{attribute 'conditionalshow'}
FUNCTION_BLOCK FB_GantryXYZ EXTENDS FB_PackML_BaseModule IMPLEMENTS I_GantryConfigProvider
VAR
	
	fbHomeMcQ           : MC_Home;
    // =========================================================
    //  DEPENDENCIES & SUB-MODULES
    // =========================================================
    _RecipeBuilder      : I_RecipeBuilder;
    ipSubModules_Init   : ARRAY[1..Parameters_PackML_Base.MAX_NO_OF_SUBMODULES] OF I_PackML_BaseModule := [];

	ExecutorCutX 		: FB_Exec_Pneumatic_PTP;
	ExecutorCutY 		: FB_Exec_Pneumatic_PTP;	
	ExecutorGrooveXY	: FB_Exec_Spindle_PTP;
	ExecutorDrill 		: FB_Exec_Drill_PTP;
	ExecTangentialFeed	: FB_Exec_Tangential_FeedTable;
	
	ExecutorNCI 		: FB_Exec_Spindle_GCodeXYZ;
	
	_Limits : ST_GantryXYZ_Limits;


    // =========================================================
    //  HMI & COMMANDS
    // =========================================================
    GantryXYZ_HMI       : ST_GantryXYZ_HMI;
    _ProgramIdRequested : E_RecipeID;

    // =========================================================
    //  COMPONENTS (AXES & CYLINDERS)
    // =========================================================
    AxisX               : FB_Component_BasicAxis := (Name := 'AxisX');
    AxisY               : FB_Component_BasicAxis := (Name := 'AxisY');
    AxisZ               : FB_Component_BasicAxis := (Name := 'AxisZ');
	AxisQ               : FB_Component_BasicAxis := (Name := 'AxisQ Tangential'); 
	
	
	NciChannel          	: FB_NciChannel := (Name := 'NCI Channel 1');
	NciChannelTangential	: FB_NciChannelTangential := (Name := 'NCI Channel Tangential');
	
	
	
	// [Typ osi: 1=X, 2=Y, 3=Z] , [Typ profilu z Enuma]
	ProfilesX : ARRAY[E_MachineProfile.eHoming..E_MachineProfile.eManual] OF ST_AxisProfile;
	ProfilesY : ARRAY[E_MachineProfile.eHoming..E_MachineProfile.eManual] OF ST_AxisProfile;
	ProfilesZ : ARRAY[E_MachineProfile.eHoming..E_MachineProfile.eManual] OF ST_AxisProfile;
	ProfilesQ : ARRAY[E_MachineProfile.eHoming..E_MachineProfile.eManual] OF ST_AxisProfile;
	
	// Flagi określające typ napędu dla konkretnej osi (TRUE = SoE/AX5000, FALSE = CoE)
    AxisX_IsSoE : BOOL := FALSE;
    AxisY_IsSoE : BOOL := FALSE;
    AxisZ_IsSoE : BOOL := FALSE;
 
	CylinderCuttingX : FB_Cylinder := (Name := 'Cylinder X');
    CylinderCuttingY : FB_Cylinder := (Name := 'Cylinder Y');

    // =========================================================
    //  HOMING STRATEGIES
    // =========================================================
    fbHomeStratX        : FB_Homing_StandardNC;
    fbHomeStratY        : FB_Homing_StandardNC;
    fbHomeStratZ        : FB_Homing_StandardNC;
	fbHomeStratQ 		: FB_Homing_Direct;

    // =========================================================
    //  ALARMS
    // =========================================================
    GantryAlarms        : ARRAY[1..GANTRY_ALARM_COUNT] OF FB_TcAlarm;
	
	ResetStratX : FB_ResetRoutine_SoEDrive;
	ResetStratY : FB_ResetRoutine_SoEDrive;
	ResetStratZ : FB_ResetRoutine_SoEDrive;

END_VAR

VAR CONSTANT
    GANTRY_ALARM_COUNT  : INT := 5;
END_VAR

METHOD PROTECTED Aborting
VAR
    i               : UDINT;
    SubModulesReady : BOOL := TRUE;
END_VAR
VAR_INST
    AbortStepTimer  : TON; 
END_VAR
CASE _CurrentMode OF

//=================================PRODUCTION MODE==================================
// POUs/GantryXYZ/FB_GantryXYZ.TcPOU -> Metoda Aborting

E_PMLUnitMode.ePMLUnitMode_Production:
    CASE SequenceState OF
        0:
            NoStateTasksToComplete := FALSE;
            
            // Logujemy rozpoczęcie procedury Abort
            ADSLOGSTR(ADSLOG_MSGTYPE_HINT, 'Aborting [0]: Zatrzymywanie kanałów i resetowanie błędów NCI...', '');
            
            NciChannel.Stop();
            NciChannelTangential.Stop();
            
            NciChannel.ResetChannel();
            NciChannelTangential.ResetChannel(); 

            AbortStepTimer(IN:=FALSE);
            SequenceState := 10;

        10:
            AbortStepTimer(IN:=TRUE, PT:=T#300MS); 
            IF AbortStepTimer.Q THEN
                AbortStepTimer(IN:=FALSE);
                
                ADSLOGSTR(ADSLOG_MSGTYPE_HINT, 'Aborting [10]: Nakazano rozpięcie (Ungroup) grup 4 i 5.', '');
                
                NciChannel.Ungroup();
                NciChannelTangential.Ungroup(); 
                SequenceState := 20;
            END_IF

        20:
            // Sprawdzanie warunku z logowaniem co jakiś czas (jeśli utknie)
            IF NOT NciChannel.IsGrouped AND NOT NciChannelTangential.IsGrouped THEN
                
                ADSLOGSTR(ADSLOG_MSGTYPE_HINT, 'Aborting [20]: Grupy rozpięte. Wyłączanie napędów i zwalnianie executorów.', '');

                AxisX.Disable();
                AxisY.Disable();
                AxisZ.Disable();
                AxisQ.Disable(); 
        
                IO.SpindleEnable := FALSE;
                IO.CoolingEnable := FALSE;
                
                CylinderCuttingX.Retract();
                CylinderCuttingY.Retract();
        
                fbHomeStratX.Abort();
                fbHomeStratY.Abort();
                fbHomeStratZ.Abort();
				fbHomeStratQ.Abort();
                
                ExecutorCutX.Abort();
                ExecutorCutY.Abort();
                ExecutorGrooveXY.Abort();
                ExecutorNCI.Abort();
                ExecTangentialFeed.Abort();
				ExecutorDrill.Abort();
                
                SequenceState := 30;
            END_IF
    
        30:
            ADSLOGSTR(ADSLOG_MSGTYPE_HINT, 'Aborting [30]: Procedura Abort zakończona sukcesem.', '');
            StateTasksComplete := TRUE;
            
    END_CASE

	//=================================MAINTENANCE & MANUAL MODE==================================
	E_PMLUnitMode.ePMLUnitMode_Maintenance, E_PMLUnitMode.ePMLUnitMode_Manual:

	CASE SequenceState OF
    
		0:
			NoStateTasksToComplete := FALSE;
			SequenceState          := SequenceState + 10;
		
		10:
			AxisX.Disable();
			AxisY.Disable();
			AxisZ.Disable();
			
			CylinderCuttingX.Retract();
			CylinderCuttingY.Retract();
			
			IO.CoolingEnable := FALSE;
			IO.SpindleEnable := FALSE;
	
			SequenceState := SequenceState + 10;
		
		20:
			StateTasksComplete := TRUE;

	END_CASE
	
END_CASE

SUPER^.Aborting();
END_METHOD

METHOD ApplyProfile
VAR_INPUT
	RequestedProfile : E_MachineProfile;
END_VAR
AxisX.WriteParameter(MC_AxisParameter.AxisMinSoftPosLimit, ProfilesX[RequestedProfile].SoftLimitMin);
AxisX.WriteParameter(MC_AxisParameter.AxisMaxSoftPosLimit, ProfilesX[RequestedProfile].SoftLimitMax);
AxisX.Acceleration := ProfilesX[RequestedProfile].Acceleration;
AxisX.Deceleration := ProfilesX[RequestedProfile].Deceleration;
AxisX.Jerk         := ProfilesX[RequestedProfile].Jerk;


AxisY.WriteParameter(MC_AxisParameter.AxisMinSoftPosLimit, ProfilesY[RequestedProfile].SoftLimitMin);
AxisY.WriteParameter(MC_AxisParameter.AxisMaxSoftPosLimit, ProfilesY[RequestedProfile].SoftLimitMax);
AxisY.Acceleration := ProfilesY[RequestedProfile].Acceleration;
AxisY.Deceleration := ProfilesY[RequestedProfile].Deceleration;
AxisY.Jerk         := ProfilesY[RequestedProfile].Jerk;


AxisZ.WriteParameter(MC_AxisParameter.AxisMinSoftPosLimit, ProfilesZ[RequestedProfile].SoftLimitMin);
AxisZ.WriteParameter(MC_AxisParameter.AxisMaxSoftPosLimit, ProfilesZ[RequestedProfile].SoftLimitMax);
AxisZ.Acceleration := ProfilesZ[RequestedProfile].Acceleration;
AxisZ.Deceleration := ProfilesZ[RequestedProfile].Deceleration;
AxisZ.Jerk         := ProfilesZ[RequestedProfile].Jerk;


AxisQ.WriteParameter(MC_AxisParameter.AxisMinSoftPosLimit, ProfilesQ[RequestedProfile].SoftLimitMin);
AxisQ.WriteParameter(MC_AxisParameter.AxisMaxSoftPosLimit, ProfilesQ[RequestedProfile].SoftLimitMax);
AxisQ.Acceleration := ProfilesQ[RequestedProfile].Acceleration;
AxisQ.Deceleration := ProfilesQ[RequestedProfile].Deceleration;
AxisQ.Jerk         := ProfilesQ[RequestedProfile].Jerk;
AxisQ.Velocity	   := ProfilesQ[RequestedProfile].Velocity;
END_METHOD

METHOD PROTECTED Clearing
VAR
	i				: UDINT;
	SubModulesReady : BOOL := TRUE;
END_VAR
VAR_INST
    LogTimer        : TON; // Timer do opóźniania logów, żeby nie zaspamować konsoli
END_VAR
CASE SequenceState OF
    0:
        NoStateTasksToComplete := FALSE;
        SequenceState          := SequenceState + 10;
    10:
		AxisX.Reset();
		AxisY.Reset();
		AxisZ.Reset();
        AxisQ.Reset(); 
		AxisX.Axis.PlcToNc.ExtSetPos := 2;
		AxisY.Axis.PlcToNc.ExtSetPos := 2;
		
        
        NciChannel.ResetChannel();
        NciChannelTangential.ResetChannel();

		SequenceState := SequenceState + 10;
		
    20:
        StateTasksComplete := TRUE;
END_CASE

SUPER^.Clearing();


LogTimer(IN := (SequenceState = 20), PT := T#2S);

IF LogTimer.Q THEN
    LogTimer(IN := FALSE); 
    
    IF AxisQ.Error THEN
        ADSLOGDINT(ADSLOG_MSGTYPE_ERROR, 'CLEARING BLOCKED BY: AxisQ! ErrorID: %d', UDINT_TO_DINT(AxisQ.ErrorID));
    END_IF
    
    IF NciChannelTangential.ChannelError THEN
        ADSLOGDINT(ADSLOG_MSGTYPE_ERROR, 'CLEARING BLOCKED BY: NciChannelTangential! ErrorID: %d', UDINT_TO_DINT(NciChannelTangential.ChannelErrorId));
    END_IF
    
    IF NciChannel.ChannelError THEN
        ADSLOGDINT(ADSLOG_MSGTYPE_ERROR, 'CLEARING BLOCKED BY: NciChannel! ErrorID: %d', UDINT_TO_DINT(NciChannel.ChannelErrorId));
    END_IF
END_IF
END_METHOD

PROPERTY Config : ST_GantryXYZ_Config
GET
Config := GantryXYZ_HMI.Config;
END_GET
SET
GantryXYZ_HMI.Config.CutterXOffsetX   := LIMIT(_Limits.CutterXOffsetX.MinVal, Config.CutterXOffsetX, _Limits.CutterXOffsetX.MaxVal);
GantryXYZ_HMI.Config.CutterXOffsetY   := LIMIT(_Limits.CutterXOffsetY.MinVal, Config.CutterXOffsetY, _Limits.CutterXOffsetY.MaxVal);
GantryXYZ_HMI.Config.CutterYOffsetX   := LIMIT(_Limits.CutterYOffsetX.MinVal, Config.CutterYOffsetX, _Limits.CutterYOffsetX.MaxVal);
GantryXYZ_HMI.Config.CutterYOffsetY   := LIMIT(_Limits.CutterYOffsetY.MinVal, Config.CutterYOffsetY, _Limits.CutterYOffsetY.MaxVal);
GantryXYZ_HMI.Config.CuttingSpeedXY  := LIMIT(_Limits.CuttingSpeedXY.MinVal, Config.CuttingSpeedXY, _Limits.CuttingSpeedXY.MaxVal);

GantryXYZ_HMI.Config.GroovingSpeedXY := LIMIT(_Limits.GroovingSpeedXY.MinVal, Config.GroovingSpeedXY, _Limits.GroovingSpeedXY.MaxVal);
GantryXYZ_HMI.Config.GroovingSpeedZ  := LIMIT(_Limits.GroovingSpeedZ.MinVal, Config.GroovingSpeedZ, _Limits.GroovingSpeedZ.MaxVal);
GantryXYZ_HMI.Config.GroovingSpeedZ   := LIMIT(_Limits.GroovingSpeedZ.MinVal, Config.GroovingSpeedZ, _Limits.GroovingSpeedZ.MaxVal);

GantryXYZ_HMI.Config.RapidSpeedX      := LIMIT(_Limits.RapidSpeedX.MinVal, Config.RapidSpeedX, _Limits.RapidSpeedX.MaxVal);
GantryXYZ_HMI.Config.RapidSpeedY      := LIMIT(_Limits.RapidSpeedY.MinVal, Config.RapidSpeedY, _Limits.RapidSpeedY.MaxVal);
GantryXYZ_HMI.Config.RapidSpeedZ      := LIMIT(_Limits.RapidSpeedZ.MinVal, Config.RapidSpeedZ, _Limits.RapidSpeedZ.MaxVal);

GantryXYZ_HMI.Config.CuttingIdleTime  := LIMIT(_Limits.CuttingIdleTime.MinVal, Config.CuttingIdleTime, _Limits.CuttingIdleTime.MaxVal);
GantryXYZ_HMI.Config.GroovingIdleTime := LIMIT(_Limits.GroovingIdleTime.MinVal, Config.GroovingIdleTime, _Limits.GroovingIdleTime.MaxVal);

GantryXYZ_HMI.Config.GlobalOffsetX := LIMIT(_Limits.GlobalOffsetX.MinVal, Config.GlobalOffsetX, _Limits.GlobalOffsetX.MaxVal);
GantryXYZ_HMI.Config.GlobalOffsetY := LIMIT(_Limits.GlobalOffsetY.MinVal, Config.GlobalOffsetY, _Limits.GlobalOffsetY.MaxVal);
GantryXYZ_HMI.Config.GlobalOffsetZ := LIMIT(_Limits.GlobalOffsetZ.MinVal, Config.GlobalOffsetZ, _Limits.GlobalOffsetZ.MaxVal);
GantryXYZ_HMI.Config.RawBoardX     := LIMIT(_Limits.RawBoardX.MinVal, Config.RawBoardX, _Limits.RawBoardX.MaxVal);
GantryXYZ_HMI.Config.RawBoardY     := LIMIT(_Limits.RawBoardY.MinVal, Config.RawBoardY, _Limits.RawBoardY.MaxVal);
GantryXYZ_HMI.Config.RawBoardZ      := LIMIT(_Limits.RawBoardZ.MinVal, Config.RawBoardZ, _Limits.RawBoardZ.MaxVal);
GantryXYZ_HMI.Config.SafeClearanceZ := LIMIT(_Limits.SafeClearanceZ.MinVal, Config.SafeClearanceZ, _Limits.SafeClearanceZ.MaxVal);

GantryXYZ_HMI.Config.RapidSpeedQ := LIMIT(_Limits.RapidSpeedQ.MinVal, Config.RapidSpeedQ, _Limits.RapidSpeedQ.MaxVal);

GantryXYZ_HMI.Config.AxisQ_SavedPos := Config.AxisQ_SavedPos;
END_SET
END_PROPERTY

METHOD PROTECTED CreateEvents
VAR_INPUT
END_VAR
// Add your event creation here
F_CreateAllEventsInClass(Alarms     := GantryAlarms,
                         ClassSize  := SIZEOF(TC_EVENTS.Gantry),
                         pInitEvent := ADR(TC_EVENTS.Gantry.InitReferenceEvent),
                         Prefix     := _Name);

// Super call to base
SUPER^.CreateEvents();
END_METHOD

METHOD CyclicLogic
VAR_INPUT
END_VAR
IF NOT _InitComplete THEN
    _InitComplete := Initialize();
    RETURN;
END_IF



SUPER^.CyclicLogic();

fbHomeStratX.bSensorInput := IO.ProximitySensorX;
fbHomeStratY.bSensorInput := IO.ProximitySensorY;
fbHomeStratZ.bSensorInput := IO.ProximitySensorZ;

fbHomeStratX.RapidVelocity := GantryXYZ_HMI.Config.RapidSpeedX;
fbHomeStratY.RapidVelocity := GantryXYZ_HMI.Config.RapidSpeedY;

fbHomeStratZ.RapidVelocity := GantryXYZ_HMI.Config.RapidSpeedZ;
//Axis Z needs to be homed always, because doesn't have an encoder 
fbHomeStratZ.bForceHoming := TRUE;

fbHomeStratX.CyclicLogic();
fbHomeStratY.CyclicLogic();
fbHomeStratZ.CyclicLogic();
fbHomeStratQ.CyclicLogic();

NciChannel.CyclicLogic();

ExecutorCutX.CyclicLogic();
ExecutorCutY.CyclicLogic();
ExecutorGrooveXY.CyclicLogic();
ExecutorNCI.CyclicLogic();
ExecTangentialFeed.CyclicLogic();
ExecutorDrill.CyclicLogic();

//Set the current alarm severity for this module
_CurrentAlarmSeverity := F_GetMaxSeverityRaised(Alarms := GantryAlarms, CurrentSeverity := _CurrentAlarmSeverity);

// Śledzenie i zapamiętywanie pozycji osi Q dla noża tangencjalnego
IF AxisQ.Axis.Status.Homed THEN 
    GantryXYZ_HMI.Config.AxisQ_SavedPos := AxisQ.Axis.NcToPlc.ActPos;
//	fbHomeStratQ.ReferencePosition := GantryXYZ_HMI.Config.AxisQ_SavedPos;
END_IF
END_METHOD

METHOD PROTECTED Execute
VAR
    localConfig : ST_RecipeBuilder_Config; // Zmienna pomocnicza dla kompilatora
END_VAR
CASE _CurrentMode OF

    //=================================PRODUCTION MODE==================================
    E_PMLUnitMode.ePMLUnitMode_Production:
        CASE SequenceState OF
            0:
                NoStateTasksToComplete := FALSE;
                // LOG: Start sekwencji
                ADSLOGSTR(ADSLOG_MSGTYPE_HINT, 'MainSeq: Rozpoczynam nowa sekwencje produkcyjna', '');
                SequenceState := 10;
                
            10: 
                SequenceState := 20;
                
			20: 
				IF _RecipeBuilder <> 0 THEN
					
					// Zależność dla FeedTable
					IF _RecipeBuilder.ExecutionRoute = E_ExecutionRoute.eFeedTable THEN
						_RecipeBuilder.GeometryWriter := ExecTangentialFeed;
					END_IF
					
					// 1. PO PROSTU KAZEMY RECEPCIE PRACOWAĆ (nie sprawdzamy co zwraca funkcja!)
					_RecipeBuilder.Build();
					
					// 2. SPRAWDZAMY FLAGI STANU
					IF _RecipeBuilder.Done THEN 
						
						// ========================================================
						// SUKCES - ROZWIDLENIE DLA FAZY 1
						// ========================================================
						localConfig := _RecipeBuilder.Config;
						
						CASE _RecipeBuilder.ExecutionRoute OF
							E_ExecutionRoute.ePTP:
								ADSLOGSTR(ADSLOG_MSGTYPE_HINT, 'MainSeq: Start Fazy 1 - Tryb PTP', '');
								SequenceState := 30; 
								
							E_ExecutionRoute.eGCode:
								ADSLOGSTR(ADSLOG_MSGTYPE_HINT, 'MainSeq: Start Fazy 1 - Tryb G-Code', '');
								SequenceState := 40;                             
								
							E_ExecutionRoute.eFeedTable:
								ADSLOGSTR(ADSLOG_MSGTYPE_HINT, 'MainSeq: Start Fazy 1 - Tryb FeedTable', '');
								SequenceState := 60; 
						END_CASE
						
					ELSIF _RecipeBuilder.Error THEN
						
						// ========================================================
						// PORAŻKA 
						// ========================================================
						ADSLOGSTR(ADSLOG_MSGTYPE_ERROR, 'MainSeq: Krok 20 - Recepta zglosila ERROR!', '');
						RaiseAlarmWithStrings(GantryAlarms[1], 'Blad budowania recepty! Sprawdz wymiary z HMI.', '');
						ChangeState(E_PMLCommand.ePMLCommand_Abort);
						SequenceState := 999;
			
					END_IF
					// Jeśli nie jest ani Done, ani Error, to maszyna po prostu nic nie robi 
					// i przechodzi do następnego cyklu PLC, dając recepcie czas na pracę (bo flaga _Busy jest aktywna).
			
				ELSE
					// Brak buildera = zły numer programu
					ADSLOGSTR(ADSLOG_MSGTYPE_ERROR, 'MainSeq: BLAD KRYTYCZNY! Brak obiektu _RecipeBuilder.', '');
					ChangeState(E_PMLCommand.ePMLCommand_Abort);
					SequenceState := 999;
				END_IF

            // ========================================================
            // FAZA 1: NARZĘDZIE GŁÓWNE
            // ========================================================
            
            // --- 1A: Wykonanie w trybie PTP (np. GrooveXY) ---
            30: 
                IF ExecutorGrooveXY.Execute() THEN SequenceState := 35; END_IF
            35: 
                IF ExecutorGrooveXY.Done THEN 
                    SequenceState := 70; 
                ELSIF ExecutorGrooveXY.Error THEN
                    RaiseAlarmWithStrings(GantryAlarms[1], 'Blad w Executorze PTP', '');
                    ChangeState(E_PMLCommand.ePMLCommand_Abort);
                    SequenceState := 999;
                END_IF
                
            // --- 1B: Wykonanie w trybie G-Code ---
            40:
                IF ExecutorNCI.Execute() THEN SequenceState := 45; END_IF
            45:
                IF ExecutorNCI.Done THEN 
                    SequenceState := 70;
                ELSIF ExecutorNCI.Error THEN
                    RaiseAlarmWithStrings(GantryAlarms[1], 'Krytyczny Blad NCI G-Code', '');
                    ChangeState(E_PMLCommand.ePMLCommand_Abort);
                    SequenceState := 999; 
                END_IF
                
            // --- 1C: Wykonanie w trybie FeedTable ---
            60:
                IF ExecTangentialFeed.Execute() THEN SequenceState := 65; END_IF
            65:
                IF ExecTangentialFeed.Done THEN 
                    SequenceState := 70;
                ELSIF ExecTangentialFeed.Error THEN
                    RaiseAlarmWithStrings(GantryAlarms[1], 'Krytyczny Blad NCI FeedTable', '');
                    ChangeState(E_PMLCommand.ePMLCommand_Abort);
                    SequenceState := 999; 
                END_IF

				
			// ========================================================
			// FAZA 1.5: WIERCENIE OTWORÓW (Opcjonalne dla każdej recepty)
			// ========================================================
			70:
				IF ExecutorDrill.Execute() THEN 
					ADSLOGSTR(ADSLOG_MSGTYPE_HINT, 'MainSeq: Faza 1.5 - Start operacji wiercenia otworów', '');
					SequenceState := 75;
				END_IF
			75:
				IF ExecutorDrill.Done THEN 
					SequenceState := 100; // Sukces -> Przejście do Fazy 2 (Docinki pneumatyczne)
				ELSIF ExecutorDrill.Error THEN
					RaiseAlarmWithStrings(GantryAlarms[1], 'Krytyczny Blad Executora Wiercenia', '');
					ChangeState(E_PMLCommand.ePMLCommand_Abort);
					SequenceState := 999; 
				END_IF	
				
				

            // ========================================================
            // FAZA 2: DOCINKA PNEUMATYCZNA (Wspólna dla wszystkich)
            // ========================================================
            100: 
                IF ExecutorCutY.Execute() THEN 
                    ADSLOGSTR(ADSLOG_MSGTYPE_HINT, 'MainSeq: Faza 2 - Start operacji CutY', '');
                    SequenceState := 110; 
                END_IF
            110: 
                IF ExecutorCutY.Done THEN 
                    SequenceState := 120;
                ELSIF ExecutorCutY.Error THEN
                    RaiseAlarmWithStrings(GantryAlarms[1], 'Blad w CutY', '');
                    ChangeState(E_PMLCommand.ePMLCommand_Abort);
                    SequenceState := 999;
                END_IF
                
            120: 
                IF ExecutorCutX.Execute() THEN 
                    ADSLOGSTR(ADSLOG_MSGTYPE_HINT, 'MainSeq: Faza 2 - Start operacji CutX', '');
                    SequenceState := 130; 
                END_IF
            130: 
                IF ExecutorCutX.Done THEN 
                    SequenceState := 1000; // Koniec całego detalu!
                ELSIF ExecutorCutX.Error THEN
                    RaiseAlarmWithStrings(GantryAlarms[1], 'Blad w CutX', '');
                    ChangeState(E_PMLCommand.ePMLCommand_Abort);
                    SequenceState := 999;
                END_IF

            // ========================================================
            // MARTWY KROK DLA BŁĘDÓW
            // ========================================================
            999:
                // Maszyna po prostu tu czeka.
                // W tle PackML przetworzy komendę ChangeState i brutalnie przerwie
                // metodę Execute(), przeskakując do metody Aborting()!
                ;
    
            // ========================================================
            // KONIEC OBRÓBKI 
            // ========================================================
            1000:            
                ADSLOGSTR(ADSLOG_MSGTYPE_HINT, 'MainSeq: Sekwencja produkcyjna zakonczona sukcesem.', '');
                StateTasksComplete := TRUE;
                StateComplete();

        END_CASE

    //=================================MAINTENANCE & MANUAL MODE==================================
    E_PMLUnitMode.ePMLUnitMode_Maintenance, E_PMLUnitMode.ePMLUnitMode_Manual:
        ;
END_CASE
END_METHOD

METHOD FB_init : BOOL
VAR_INPUT
	bInitRetains : BOOL; // if TRUE, the retain variables are initialized (warm start / cold start)
	bInCopyCode : BOOL;  // if TRUE, the instance afterwards gets moved into the copy code (online change)
END_VAR



// ===============================================================================
// LIMIT COMMITTED FROM HMI
// ===============================================================================
_Limits.CutterXOffsetX.MinVal := -200.0;   _Limits.CutterXOffsetX.MaxVal := 200.0;
_Limits.CutterXOffsetY.MinVal := -200.0;   _Limits.CutterXOffsetY.MaxVal := 200.0;
_Limits.CutterYOffsetX.MinVal := -200.0;   _Limits.CutterYOffsetX.MaxVal := 200.0;
_Limits.CutterYOffsetY.MinVal := -200.0;   _Limits.CutterYOffsetY.MaxVal := 200.0;
_Limits.GlobalOffsetX.MinVal   := -500.0;   _Limits.GlobalOffsetX.MaxVal   := 500.0;
_Limits.GlobalOffsetY.MinVal   := -500.0;   _Limits.GlobalOffsetY.MaxVal   := 500.0;
_Limits.GlobalOffsetZ.MinVal   := -5.0;     _Limits.GlobalOffsetZ.MaxVal   := 5.0;
_Limits.CuttingSpeedXY.MinVal  := 1.0;     _Limits.CuttingSpeedXY.MaxVal  := 100.0;
_Limits.GroovingSpeedXY.MinVal := 1.0;     _Limits.GroovingSpeedXY.MaxVal := 100.0;
_Limits.GroovingSpeedZ.MinVal  := 1.0;     _Limits.GroovingSpeedZ.MaxVal  := 100.0;
_Limits.RapidSpeedX.MinVal     := 1.0;     _Limits.RapidSpeedX.MaxVal     := 200.0;
_Limits.RapidSpeedY.MinVal     := 1.0;     _Limits.RapidSpeedY.MaxVal     := 200.0;
_Limits.RapidSpeedZ.MinVal     := 1.0;     _Limits.RapidSpeedZ.MaxVal     := 20.0;
_Limits.CuttingIdleTime.MinVal  := 0.0;    _Limits.CuttingIdleTime.MaxVal  := 10.0;
_Limits.GroovingIdleTime.MinVal := 0.0;    _Limits.GroovingIdleTime.MaxVal := 10.0;
_Limits.RawBoardX.MinVal       := 200.0;   _Limits.RawBoardX.MaxVal       := 1220.0;
_Limits.RawBoardY.MinVal       := 200.0;   _Limits.RawBoardY.MaxVal       := 2440.0;
_Limits.RawBoardZ.MinVal       := 1.0;     _Limits.RawBoardZ.MaxVal       := 12.0;
_Limits.SafeClearanceZ.MinVal  := 1.0;     _Limits.SafeClearanceZ.MaxVal  := 100.0;
_Limits.RapidSpeedQ.MinVal 	   := 1.0; 	   _Limits.RapidSpeedQ.MaxVal := 1080.0; 


InitProfiles();
END_METHOD

// Provides interlocks for HMI control and updates HMI status information for this module
//Only in this place HMI input can overwrite internal data 
METHOD PROTECTED HMICommunication
// This method is called cyclically by CyclicLogic()
SUPER^.HMICommunication();

_ProgramIdRequested   := GantryXYZ_HMI.Command.ProgramIdRequested;

GantryXYZ_HMI.Limits := _Limits;
THIS^.Config := GantryXYZ_HMI.Config;
END_METHOD

METHOD PROTECTED HMIPermissions
//General Mode Based Monitoring and handling of HMI control
CASE _CurrentMode OF
   
 E_PMLUnitMode.ePMLUnitMode_Production:
        CASE _CurrentState OF
            E_PMLState.ePMLState_Stopped:
				AllowHMIControl(ThisModuleOnly := FALSE);
            E_PMLState.ePMLState_Idle:
				AllowHMIControl(ThisModuleOnly := FALSE);
            E_PMLState.ePMLState_Suspended:
         		AllowHMIControl(ThisModuleOnly := FALSE);
            E_PMLState.ePMLState_Execute:
            	AllowHMIControl(ThisModuleOnly := FALSE); 
            E_PMLState.ePMLState_Aborted:
                AllowHMIControl(ThisModuleOnly := FALSE); 
            E_PMLState.ePMLState_Held:
                AllowHMIControl(ThisModuleOnly := FALSE); 
            E_PMLState.ePMLState_Complete:
          		AllowHMIControl(ThisModuleOnly := FALSE); 
        END_CASE
		
    E_PMLUnitMode.ePMLUnitMode_Manual:
        AllowHMIControl(ThisModuleOnly := FALSE); 
	E_PMLUnitMode.ePMLUnitMode_Maintenance:
        AllowHMIControl(ThisModuleOnly := FALSE); 
END_CASE
END_METHOD

//! @summary Basic module initialization logic
METHOD PROTECTED Initialize : BOOL;
VAR
    i                        : UDINT;
    varInfo                  : __SYSTEM.VAR_INFO;
    AllSubUnitsInitialized   : BOOL := TRUE;
    AllComponentsInitialized : BOOL := TRUE;
END_VAR

//! @description This method is called by <c>CyclicLogic()</c> as required
Initialize := FALSE;
CASE DescendantSequenceState OF
    0:
		RegisterComponent(AxisX);
		RegisterComponent(AxisY);	
		RegisterComponent(AxisZ);
		RegisterComponent(AxisQ);	
		RegisterComponent(CylinderCuttingY);
		RegisterComponent(CylinderCuttingX);
		RegisterComponent(NciChannel);
		RegisterComponent(NciChannelTangential); 
        _LogModeChanges         := FALSE;
        _LogStateChanges        := FALSE;
		
        DescendantSequenceState := DescendantSequenceState + 10;
    10:
		// Wczytanie zapisanej pozycji dla noża tangencjalnego
		fbHomeStratQ.ReferencePosition := GantryXYZ_HMI.Config.AxisQ_SavedPos;
		
		// Przypisanie osi do strategii
		fbHomeStratX.Axis := AxisX;
		fbHomeStratY.Axis := AxisY;
		fbHomeStratZ.Axis := AxisZ;
		fbHomeStratQ.Axis := AxisQ;
		
		
		// Wstrzyknięcie strategii do osi (Dependency Injection)
		AxisX.HomeMethod := fbHomeStratX;
		AxisY.HomeMethod := fbHomeStratY;
		AxisZ.HomeMethod := fbHomeStratZ;
		AxisQ.HomeMethod := fbHomeStratQ;
		
		// Wstrzykiwanie zależności do Executora Cut X
		ExecutorCutX.CutDirection   := E_CutDirection.eCutX;
		ExecutorCutX.AxisX          := AxisX;
		ExecutorCutX.AxisY          := AxisY;
		ExecutorCutX.AxisZ          := AxisZ;
		ExecutorCutX.Cylinder       := CylinderCuttingX; // Podpinamy siłownik X!
		ExecutorCutX.ConfigProvider := THIS^;
		
		// Wstrzykiwanie zależności do Executora Cut Y 
		ExecutorCutY.CutDirection   := E_CutDirection.eCutY;
		ExecutorCutY.AxisX          := AxisX;
		ExecutorCutY.AxisY          := AxisY;
		ExecutorCutY.AxisZ          := AxisZ;
		ExecutorCutY.Cylinder       := CylinderCuttingY; // Podpinamy siłownik Y!
		ExecutorCutY.ConfigProvider := THIS^;
		
		// Wstrzykiwanie zależności do Executora NCI
		ExecutorNCI.AxisX          := AxisX;
		ExecutorNCI.AxisY          := AxisY;
		ExecutorNCI.AxisZ          := AxisZ;
		ExecutorNCI.NciChannel     := NciChannel; // Twój nowy kanał
		ExecutorNCI.ConfigProvider := THIS^;
		
		// Wstrzykiwanie zależności do ExecTangentialFeed
		ExecTangentialFeed.AxisX          := AxisX;
		ExecTangentialFeed.AxisY          := AxisY;
		ExecTangentialFeed.AxisZ          := AxisZ;
		ExecTangentialFeed.AxisQ 		  := AxisQ;
		ExecTangentialFeed.NciChannel     := NciChannelTangential; 
		ExecTangentialFeed.ConfigProvider := THIS^;
		
		// Wstrzykiwanie zależności do Executora Drill PTP
		ExecutorDrill.AxisX := AxisX;
		ExecutorDrill.AxisY := AxisY;
		ExecutorDrill.AxisZ := AxisZ;
		ExecutorDrill.AxisQ := AxisQ;
		ExecutorDrill.ConfigProvider := THIS^;
		

		// Wstrzyknięcie strategii resetu sprzętowego
		// Oś X
		IF AxisX_IsSoE THEN
			AxisX.ResetMethod := ResetStratX;
		END_IF
		
		// Oś Y
		IF AxisY_IsSoE THEN
			AxisY.ResetMethod := ResetStratY;
		END_IF
		
		// Oś Z
		IF AxisZ_IsSoE THEN
			AxisZ.ResetMethod := ResetStratZ;
		END_IF
		
		
	
		// Wstrzykiwanie zależności do Executora Groove XY
		ExecutorGrooveXY.AxisX         := AxisX;
		ExecutorGrooveXY.AxisY         := AxisY;
		ExecutorGrooveXY.AxisZ         := AxisZ;
		ExecutorGrooveXY.ConfigProvider := THIS^;
		
		// Dla zwykłego kanału
		NciChannel.stAxisIds.nX := AxisX.Axis.NcToPlc.AxisId;
		NciChannel.stAxisIds.nY := AxisY.Axis.NcToPlc.AxisId;
		NciChannel.stAxisIds.nZ := AxisZ.Axis.NcToPlc.AxisId;

		// Dla kanału tangencjalnego 
		NciChannelTangential.stAxisIds.nX  := AxisX.Axis.NcToPlc.AxisId;
		NciChannelTangential.stAxisIds.nY  := AxisY.Axis.NcToPlc.AxisId;
		NciChannelTangential.stAxisIds.nZ  := AxisZ.Axis.NcToPlc.AxisId;
		NciChannelTangential.stAxisIds.nQ1 := AxisQ.Axis.NcToPlc.AxisId;

		
        DescendantSequenceState := DescendantSequenceState + 10;
		//initialize persistent

    20:
        //Copy Mode names
        FOR i := 1 TO 3 DO
            ModeNames[i] := F_UnitModeToString(UDINT_TO_DINT(i));
        END_FOR

        DescendantSequenceState := DescendantSequenceState + 10;
    30:
        //Call the Super
        IF SUPER^.Initialize() THEN
			ReadAxisParameters();
            DescendantSequenceState := DescendantSequenceState + 10;
        END_IF
    40:
        Initialize := TRUE;
END_CASE
END_METHOD

METHOD PRIVATE InitProfiles
VAR_INPUT
END_VAR
// ===============================================================================
// PROFIL 1: HOMING (Otwarte limity do bazowania, powolne i miękkie ruchy)
// ===============================================================================
// --- OŚ X ---
ProfilesX[E_MachineProfile.eHoming].SoftLimitMin := -1250.0;
ProfilesX[E_MachineProfile.eHoming].SoftLimitMax := 1250.0;
ProfilesX[E_MachineProfile.eHoming].Acceleration := 200.0;
ProfilesX[E_MachineProfile.eHoming].Deceleration := 200.0;
ProfilesX[E_MachineProfile.eHoming].Jerk         := 500.0;

// --- OŚ Y ---
ProfilesY[E_MachineProfile.eHoming].SoftLimitMin := -2300.0;
ProfilesY[E_MachineProfile.eHoming].SoftLimitMax := 2300.0;
ProfilesY[E_MachineProfile.eHoming].Acceleration := 200.0;
ProfilesY[E_MachineProfile.eHoming].Deceleration := 200.0;
ProfilesY[E_MachineProfile.eHoming].Jerk         := 500.0;

// --- OŚ Z ---
ProfilesZ[E_MachineProfile.eHoming].SoftLimitMin := -100.0;
ProfilesZ[E_MachineProfile.eHoming].SoftLimitMax := 100.0;
ProfilesZ[E_MachineProfile.eHoming].Acceleration := 10.0;
ProfilesZ[E_MachineProfile.eHoming].Deceleration := 100.0;
ProfilesZ[E_MachineProfile.eHoming].Jerk         := 200.0;

// --- OŚ Q ---
ProfilesQ[E_MachineProfile.eHoming].SoftLimitMin := -300.0;
ProfilesQ[E_MachineProfile.eHoming].SoftLimitMax := 300.0;
ProfilesQ[E_MachineProfile.eHoming].Acceleration := 15000.0;
ProfilesQ[E_MachineProfile.eHoming].Deceleration := 15000.0;
ProfilesQ[E_MachineProfile.eHoming].Jerk         := 48322.8;


// ===============================================================================
// PROFIL 2: PRODUCTION (Wąskie limity dla bezpieczeństwa, wysoka dynamika pracy)
// ===============================================================================
// --- OŚ X ---
ProfilesX[E_MachineProfile.eProduction].SoftLimitMin := -20.0;
ProfilesX[E_MachineProfile.eProduction].SoftLimitMax := 1200.0;
ProfilesX[E_MachineProfile.eProduction].Acceleration := 1500.0;
ProfilesX[E_MachineProfile.eProduction].Deceleration := 8000.0;
ProfilesX[E_MachineProfile.eProduction].Jerk         := 15000.0;

// --- OŚ Y ---
ProfilesY[E_MachineProfile.eProduction].SoftLimitMin := -20.0;
ProfilesY[E_MachineProfile.eProduction].SoftLimitMax := 2200.0;
ProfilesY[E_MachineProfile.eProduction].Acceleration := 1500.0;
ProfilesY[E_MachineProfile.eProduction].Deceleration := 8000.0;
ProfilesY[E_MachineProfile.eProduction].Jerk         := 15000.0;

// --- OŚ Z ---
ProfilesZ[E_MachineProfile.eProduction].SoftLimitMin := -10.0;
ProfilesZ[E_MachineProfile.eProduction].SoftLimitMax := 90.0;
ProfilesZ[E_MachineProfile.eProduction].Acceleration := 10.0;
ProfilesZ[E_MachineProfile.eProduction].Deceleration := 200.0;
ProfilesZ[E_MachineProfile.eProduction].Jerk         := 300.0;

// --- OŚ Q ---
ProfilesQ[E_MachineProfile.eProduction].SoftLimitMin := -300.0;
ProfilesQ[E_MachineProfile.eProduction].SoftLimitMax := 300.0;
ProfilesQ[E_MachineProfile.eProduction].Acceleration := 15000.0;
ProfilesQ[E_MachineProfile.eProduction].Deceleration := 15000.0;
ProfilesQ[E_MachineProfile.eProduction].Jerk         := 48322.8;

// ===============================================================================
// PROFIL 3: MANUAL (Jogowanie, otwarte limity, umiarkowana dynamika dla operatora)
// ===============================================================================
// --- OŚ X ---
ProfilesX[E_MachineProfile.eManual].SoftLimitMin := -50.0;
ProfilesX[E_MachineProfile.eManual].SoftLimitMax := 1250.0;
ProfilesX[E_MachineProfile.eManual].Acceleration := 500.0;
ProfilesX[E_MachineProfile.eManual].Deceleration := 1000.0;  
ProfilesX[E_MachineProfile.eManual].Jerk         := 2000.0;

// --- OŚ Y ---
ProfilesY[E_MachineProfile.eManual].SoftLimitMin := -100.0;
ProfilesY[E_MachineProfile.eManual].SoftLimitMax := 2500.0;
ProfilesY[E_MachineProfile.eManual].Acceleration := 500.0;
ProfilesY[E_MachineProfile.eManual].Deceleration := 1000.0;
ProfilesY[E_MachineProfile.eManual].Jerk         := 2000.0;

// --- OŚ Z ---
ProfilesZ[E_MachineProfile.eManual].SoftLimitMin := -20.0;
ProfilesZ[E_MachineProfile.eManual].SoftLimitMax := 100.0;
ProfilesZ[E_MachineProfile.eManual].Acceleration := 10.0;
ProfilesZ[E_MachineProfile.eManual].Deceleration := 200.0;
ProfilesZ[E_MachineProfile.eManual].Jerk         := 300.0;

// --- OŚ Q ---
ProfilesQ[E_MachineProfile.eManual].SoftLimitMin := -300.0;
ProfilesQ[E_MachineProfile.eManual].SoftLimitMax := 300.0;
ProfilesQ[E_MachineProfile.eManual].Acceleration := 15000.0;
ProfilesQ[E_MachineProfile.eManual].Deceleration := 15000.0;
ProfilesQ[E_MachineProfile.eManual].Jerk         := 48322.8;
END_METHOD

METHOD PRIVATE IsZAboveMaterial : BOOL
VAR_INST
    MaterialTopZ : REAL;
END_VAR
MaterialTopZ := GantryXYZ_HMI.Config.GlobalOffsetZ + GantryXYZ_HMI.Config.RawBoardZ;

IF AxisZ.Axis.NcToPlc.ActPos >= MaterialTopZ THEN
    IsZAboveMaterial := TRUE;
ELSE
    IsZAboveMaterial := FALSE;
END_IF
END_METHOD

METHOD PRIVATE MoveZToSafePosition
VAR_INST
    MaterialTopZ : REAL;
    SafeZ        : REAL;
    SpeedZ       : LREAL;
END_VAR
MaterialTopZ := GantryXYZ_HMI.Config.GlobalOffsetZ + GantryXYZ_HMI.Config.RawBoardZ;
SafeZ := MaterialTopZ + GantryXYZ_HMI.Config.SafeClearanceZ;

SpeedZ := GantryXYZ_HMI.Config.RapidSpeedZ;

IF SpeedZ <= 0.0 THEN
    IF AxisZ.AxisParameters.fRefVeloSearch > 0.0 THEN
        SpeedZ := (AxisZ.AxisParameters.fRefVeloSearch);
    ELSE
        SpeedZ := 5.0;
    END_IF
END_IF

IF SafeZ <= 0.0 THEN
    SafeZ := AxisZ.AxisParameters.fEncRefPosition; 
END_IF

AxisZ.Velocity := SpeedZ;
AxisZ.MoveAbsolute(SafeZ, 0);
END_METHOD

PROPERTY ProgramIdRequested : E_RecipeID
GET
ProgramIdRequested := _ProgramIdRequested;
END_GET
SET
// Aktualizacja zmiennej wewnętrznej
_ProgramIdRequested := ProgramIdRequested;

// Aktualizacja struktury HMI, aby ramka (Frame) na wizualizacji od razu zareagowała na zmianę
GantryXYZ_HMI.Command.ProgramIdRequested := ProgramIdRequested;
END_SET
END_PROPERTY

METHOD PRIVATE ReadAxisParameters
VAR_INPUT
END_VAR
//We use it to parametrize Homing Strategies directly from the UI
IF AxisQ.AxisParameters.fRefVeloSearch > 0.0 THEN
    fbHomeStratQ.HomingVelocity := AxisQ.AxisParameters.fRefVeloSearch;
ELSE
    fbHomeStratQ.HomingVelocity := 50.0;
END_IF

IF AxisX.AxisParameters.fRefVeloSearch > 0.0 THEN
    fbHomeStratX.HomingVelocity := AxisX.AxisParameters.fRefVeloSearch;
ELSE
    fbHomeStratX.HomingVelocity := 50.0;
END_IF

IF AxisY.AxisParameters.fRefVeloSearch > 0.0 THEN
    fbHomeStratY.HomingVelocity := AxisY.AxisParameters.fRefVeloSearch;
ELSE
    fbHomeStratY.HomingVelocity := 50.0;
END_IF

IF AxisZ.AxisParameters.fRefVeloSearch > 0.0 THEN
    fbHomeStratZ.HomingVelocity := AxisZ.AxisParameters.fRefVeloSearch;
ELSE
    fbHomeStratZ.HomingVelocity := 5.0;
END_IF

fbHomeStratX.ReferencePosition := AxisX.AxisParameters.fEncRefPosition;
fbHomeStratY.ReferencePosition := AxisY.AxisParameters.fEncRefPosition;
fbHomeStratZ.ReferencePosition := AxisZ.AxisParameters.fEncRefPosition;
END_METHOD

PROPERTY RecipeBuilder : I_RecipeBuilder
GET
RecipeBuilder := _RecipeBuilder;
END_GET
SET
_RecipeBuilder := RecipeBuilder;

ExecutorCutX.RecipeBuilder := _RecipeBuilder;
ExecutorCutY.RecipeBuilder := _RecipeBuilder;
ExecutorGrooveXY.RecipeBuilder := _RecipeBuilder;
ExecutorNCI.RecipeBuilder := _RecipeBuilder;
ExecTangentialFeed.RecipeBuilder := _RecipeBuilder;
ExecutorDrill.RecipeBuilder := _RecipeBuilder;
END_SET
END_PROPERTY

PROPERTY RefAxisX : I_BasicAxis
GET
RefAxisX := AxisX;
END_GET
END_PROPERTY

METHOD PROTECTED Resetting
VAR
    i : UDINT;
    SubModulesReady : BOOL := TRUE;
END_VAR
VAR_INST
    DelayTimer : TON;
END_VAR
CASE _CurrentMode OF

    E_PMLUnitMode.ePMLUnitMode_Production:
        CASE SequenceState OF
            0:
                NoStateTasksToComplete := FALSE;
                StateTasksComplete     := FALSE;
                SequenceState          := 10;
				DelayTimer(IN := FALSE);
        
            10:
                AxisX.Enable();
                AxisY.Enable();
                AxisZ.Enable();
                AxisQ.Enable();
                SequenceState := 20;
        
            20:
                IF AxisX.Enabled AND AxisY.Enabled AND AxisZ.Enabled AND AxisQ.Enabled THEN
                    SequenceState := 25;
                END_IF
        
			25:
				IF NOT AxisZ.Busy THEN
					IF AxisZ.Axis.Status.Homed THEN
						IF NOT IsZAboveMaterial() THEN
							MoveZToSafePosition();
							DelayTimer(IN := FALSE);
							SequenceState := 27;
						ELSE
							SequenceState := 30;
						END_IF
					ELSE
						SequenceState := 30;
					END_IF
				END_IF
            27:
                IF AxisZ.InPosition THEN
                    SequenceState := 30;
                ELSIF AxisZ.Error THEN
                    SequenceState := 99;
                END_IF
                
            30:   
                fbHomeStratQ.Execute();
                DelayTimer(IN := TRUE, PT := T#700MS);
                IF DelayTimer.Q THEN
                    DelayTimer(IN := FALSE); 
                    SequenceState := 31;
                END_IF
				
			31:	
				IF fbHomeStratQ.Done THEN
                    SequenceState := 32;
				END_IF	
			
			32: 
		    	fbHomeStratZ.Execute();
                DelayTimer(IN := TRUE, PT := T#700MS);
                IF DelayTimer.Q THEN
                    DelayTimer(IN := FALSE); 
                    SequenceState := 34;
                END_IF

            34:     
				fbHomeStratY.Execute();    
                DelayTimer(IN := TRUE, PT := T#700MS);
                IF DelayTimer.Q THEN
                    DelayTimer(IN := FALSE); 
                    SequenceState := 38;
                END_IF


            38: 
				fbHomeStratX.Execute();    
                DelayTimer(IN := TRUE, PT := T#700MS);
                IF DelayTimer.Q THEN
                    DelayTimer(IN := FALSE); 
                    SequenceState := 44;
                END_IF
				
        
			44: 	
				IF fbHomeStratX.Done AND fbHomeStratY.Done THEN
                    SequenceState := 50;
                ELSIF fbHomeStratX.Error OR fbHomeStratY.Error OR fbHomeStratQ.Error THEN
                    SequenceState := 99;
                END_IF
				
            50:
                StateTasksComplete := TRUE;
                SequenceState      := 0; 
        
            99:
                ChangeState(E_PMLCommand.ePMLCommand_Abort);
                
        END_CASE

    E_PMLUnitMode.ePMLUnitMode_Maintenance, E_PMLUnitMode.ePMLUnitMode_Manual:
        CASE SequenceState OF
            0:
                NoStateTasksToComplete := FALSE;
                SequenceState := 10;

            10:
                AxisX.Enable();
                AxisY.Enable();
                AxisZ.Enable();
                AxisQ.Enable();

                IF AxisX.Enabled AND AxisY.Enabled AND AxisZ.Enabled AND AxisQ.Enabled THEN
                    SequenceState := 20;
                END_IF

            20:
                StateTasksComplete := TRUE;
        END_CASE

END_CASE

SUPER^.Resetting();
END_METHOD

// Called one Cycle on State Change
METHOD PROTECTED StateChanged
VAR_INPUT
END_VAR
// Wywołujemy kod bazowy frameworka
SUPER^.StateChanged();

// Centralne zarządzanie dynamiką na podstawie nowo osiągniętego stanu maszyny!
CASE _CurrentMode OF
    
    // ==========================================
    // TRYB PRODUKCYJNY
    // ==========================================
    E_PMLUnitMode.ePMLUnitMode_Production:
        CASE _CurrentState OF
            
            E_PMLState.ePMLState_Resetting:
                // W trakcie bazowania osie mają inne limity i spokojnie przyspieszają
                ApplyProfile(E_MachineProfile.eHoming);
                

            E_PMLState.ePMLState_Starting, 
            E_PMLState.ePMLState_Execute:
                // Przed startem lub w trakcie pracy ładujemy agresywny profil produkcyjny
                ApplyProfile(E_MachineProfile.eProduction);
                
            E_PMLState.ePMLState_Aborting:
                // Gdy maszyna wpada w awarię, możemy zapiąć profil z ekstremalnie wysoką Deceleracją!
                ApplyProfile(E_MachineProfile.eProduction); // Albo stworzyć nowy profil eEmergency!
			E_PMLState.ePMLState_Stopped:
				ApplyProfile(E_MachineProfile.eHoming);				
			E_PMLState.ePMLState_Aborted:
				ApplyProfile(E_MachineProfile.eHoming);
        END_CASE
        
    // ==========================================
    // TRYB RĘCZNY / SERWISOWY
    // ==========================================
    E_PMLUnitMode.ePMLUnitMode_Manual:
	      
          CASE _CurrentState OF
            
            E_PMLState.ePMLState_Resetting:
                // W trakcie bazowania osie mają inne limity i spokojnie przyspieszają
                ApplyProfile(E_MachineProfile.eHoming);
                
            E_PMLState.ePMLState_Starting, 
            E_PMLState.ePMLState_Execute:
                // Przed startem lub w trakcie pracy ładujemy agresywny profil produkcyjny
                ApplyProfile(E_MachineProfile.eProduction);
                
            E_PMLState.ePMLState_Aborting:
                // Gdy maszyna wpada w awarię, możemy zapiąć profil z ekstremalnie wysoką Deceleracją!
                ApplyProfile(E_MachineProfile.eProduction); // Albo stworzyć nowy profil eEmergency!
			E_PMLState.ePMLState_Aborted:
				ApplyProfile(E_MachineProfile.eHoming);
				
			E_PMLState.ePMLState_Stopped:
				ApplyProfile(E_MachineProfile.eHoming);	
                
        END_CASE
    E_PMLUnitMode.ePMLUnitMode_Maintenance:
        
      
        CASE _CurrentState OF
            
            E_PMLState.ePMLState_Resetting:
                // W trakcie bazowania osie mają inne limity i spokojnie przyspieszają
                ApplyProfile(E_MachineProfile.eHoming);
                
            E_PMLState.ePMLState_Starting, 
            E_PMLState.ePMLState_Execute:
                // Przed startem lub w trakcie pracy ładujemy agresywny profil produkcyjny
                ApplyProfile(E_MachineProfile.eProduction);
                
            E_PMLState.ePMLState_Aborting:
                // Gdy maszyna wpada w awarię, możemy zapiąć profil z ekstremalnie wysoką Deceleracją!
                ApplyProfile(E_MachineProfile.eProduction); // Albo stworzyć nowy profil eEmergency!
				
			E_PMLState.ePMLState_Aborted:
				ApplyProfile(E_MachineProfile.eHoming);
			
			E_PMLState.ePMLState_Stopped:
				ApplyProfile(E_MachineProfile.eHoming);	
                
        END_CASE
END_CASE
END_METHOD

END_FUNCTION_BLOCK

(* stored: Version 1.1.0.1, ProductVersion 3.1.4024.15
   POU FB_GantryXYZ: Id {474e1990-f731-0ed9-052c-42626742a38f}, SpecialFunc None
   Folder Properties: Id {b05cc7e1-dc37-4910-986a-f085b4a0163d}
   Folder States: Id {8df42c9b-c051-49f1-9767-900503632339}
   Method Aborting: Id {5476dfef-6652-4e6b-8928-3724a50553de}
   Method ApplyProfile: Id {4f1c09f3-f65c-4d5f-b754-c9973148d42b}
   Method Clearing: Id {9be5800b-bdc3-471f-9b7d-42ef121d5c77}
   Property Config: Id {ca63134f-ae96-41d5-9585-0ef3c006e9b8}
   Get Get: Id {076a1a2b-8400-4320-936d-862f5092941b}
   Set Set: Id {f4f87703-cd5d-4c7f-91bc-6d612ff58e00}
   Method CreateEvents: Id {40e5a283-7f33-033f-0879-cc11ecabc43d}
   Method CyclicLogic: Id {0cfbfa67-40d6-05d6-0515-ef1c50353a78}
   Method Execute: Id {895d1ef9-5e85-47dd-a8bf-b32885837641}
   Method FB_init: Id {8fe58202-5a1a-4ae0-a78e-7b540fc3cb9d}
   Method HMICommunication: Id {0dce72f4-da14-4dd2-b6a3-5db9db3404e0}
   Method HMIPermissions: Id {a7a517c4-9176-4ef6-9045-d889c05c8a21}
   Method Initialize: Id {ba85f303-ffbe-03ad-229b-3741bd93e6e2}
   Method InitProfiles: Id {e8f6b23a-e3a6-49b3-8534-441f1020eeeb}
   Method IsZAboveMaterial: Id {51c33e2d-9980-4bce-a548-57fca5c8ab84}
   Method MoveZToSafePosition: Id {acabef9e-913d-43a5-abe7-a6cc0b93fa0e}
   Property ProgramIdRequested: Id {3b163a54-6fcd-4be2-bb98-ad529d342348}
   Get Get: Id {21210547-61ea-4bd8-a78a-96552b4742ab}
   Set Set: Id {2bb8002c-0857-45bb-b53e-f611a5c233b9}
   Method ReadAxisParameters: Id {fa8e4d08-dd4b-43dc-aa98-9f8ef932c8a4}
   Property RecipeBuilder: Id {7e3c2008-dd15-410b-92f3-2adf472e0386}
   Get Get: Id {646b66c6-cab8-496a-a121-e2412f446155}
   Set Set: Id {c356b1c0-c208-4ab6-be6c-2b4118aa8dde}
   Property RefAxisX: Id {967ef8ae-5559-4f2d-852f-051df897bca4}
   Get Get: Id {466186e1-ca25-455d-b3ae-fb439bbd9016}
   Method Resetting: Id {e7a01217-de28-430f-aeef-f83d9f1b6f0d}
   Method StateChanged: Id {3f8ec15a-7a14-4ca0-a5c1-a685d643ee3a} *)
